(* CODESYS project MyRPIEtherCAT_2ESC.project

Project tree, tasks and I/O mapping:
  Device : CODESYS Control for Raspberry Pi SL, 3S - Smart Software Solutions GmbH, version 3.5.10.20
    application TestBlink
      libraries: Standard, * (System); Util, * (System)
      task MainTask (cyclic, interval 4000 µs, priority 0) calls EtherCAT_Master.EtherCAT_Task [EtherCAT_Master.EtherCAT_Task], PLC_PRG
      program PLC_PRG [LD]
      global variables GVL
    SoftMotion General Axis Pool
    I²C
    SPI
    GPIOs_A_B : GPIOs A/B, 3S - Smart Software Solutions GmbH, version 1.1.1.10
        output TestBlink.GVL.MASTER_LED1 : BOOL  // digital outputs (GPIO0..GPIO31).Bit17
        output TestBlink.GVL.MASTER_LED2 : BOOL  // digital outputs (GPIO0..GPIO31).Bit27
        unmapped channels: digital inputs (GPIO0..GPIO31), digital outputs (GPIO0..GPIO31)
    Onewire
    Camera device
      <Empty>
    EtherCAT_Master : EtherCAT Master, 3S - Smart Software Solutions GmbH, version 3.5.10.0
        settings: SrcAddress1 = 47143; SrcAddress2 = 3943328884
      XMC_ESC : XMC_ESC, Bahoza, order no. XMC_ESC, version Revision=16#00000000
          settings: StationAlias = 1001; Optional = False; DC sync0 cycletime = 4000; DC sync1 cycletime = 4000; RxTxPdo.NumberofExcludes = 0; RxTxPdo.NumberofEntries = 12; RxTxPdo.Index = 16#1600; RxTxPdo.Fixed = True; RxTxPdo.Mandatory = True; RxTxPdo.Virtual = False; RxTxPdo.Sm = 2; RxTxPdo.Su = 2; RxTxPdo.Name = 'OUT_GENERIC process data mapping'; RxTxPdo.DependOnSlot = False; RxTxPdo.DependOnSlotGroup = False; RxTxPdo.OverwrittenByModule = False; OUT_GEN_INT1.Index = 16#7000; OUT_GEN_INT1.SubIndex = 1; OUT_GEN_INT1.Size = 16; OUT_GEN_INT1.Offset = 0; OUT_GEN_INT1.DependOnSlot = False; OUT_GEN_INT1.DependOnSlotGroup = False; OUT_GEN_INT2.Index = 16#7000; OUT_GEN_INT2.SubIndex = 2; OUT_GEN_INT2.Size = 16; OUT_GEN_INT2.Offset = 0; OUT_GEN_INT2.DependOnSlot = False; OUT_GEN_INT2.DependOnSlotGroup = False; OUT_GEN_INT3.Index = 16#7000; OUT_GEN_INT3.SubIndex = 3; OUT_GEN_INT3.Size = 16; OUT_GEN_INT3.Offset = 0; OUT_GEN_INT3.DependOnSlot = False; OUT_GEN_INT3.DependOnSlotGroup = False; OUT_GEN_INT4.Index = 16#7000; OUT_GEN_INT4.SubIndex = 4; OUT_GEN_INT4.Size = 16; OUT_GEN_INT4.Offset = 0; OUT_GEN_INT4.DependOnSlot = False; OUT_GEN_INT4.DependOnSlotGroup = False;
            OUT_GEN_Bit1.Index = 16#7000; OUT_GEN_Bit1.SubIndex = 5; OUT_GEN_Bit1.Size = 1; OUT_GEN_Bit1.Offset = 0; OUT_GEN_Bit1.DependOnSlot = False; OUT_GEN_Bit1.DependOnSlotGroup = False; OUT_GEN_Bit2.Index = 16#7000; OUT_GEN_Bit2.SubIndex = 6; OUT_GEN_Bit2.Size = 1; OUT_GEN_Bit2.Offset = 0; OUT_GEN_Bit2.DependOnSlot = False; OUT_GEN_Bit2.DependOnSlotGroup = False; OUT_GEN_Bit3.Index = 16#7000; OUT_GEN_Bit3.SubIndex = 7; OUT_GEN_Bit3.Size = 1; OUT_GEN_Bit3.Offset = 0; OUT_GEN_Bit3.DependOnSlot = False; OUT_GEN_Bit3.DependOnSlotGroup = False; OUT_GEN_Bit4.Index = 16#7000; OUT_GEN_Bit4.SubIndex = 8; OUT_GEN_Bit4.Size = 1; OUT_GEN_Bit4.Offset = 0; OUT_GEN_Bit4.DependOnSlot = False; OUT_GEN_Bit4.DependOnSlotGroup = False; OUT_GEN_Bit5.Index = 16#7000; OUT_GEN_Bit5.SubIndex = 9; OUT_GEN_Bit5.Size = 1; OUT_GEN_Bit5.Offset = 0; OUT_GEN_Bit5.DependOnSlot = False; OUT_GEN_Bit5.DependOnSlotGroup = False; OUT_GEN_Bit6.Index = 16#7000; OUT_GEN_Bit6.SubIndex = 10; OUT_GEN_Bit6.Size = 1; OUT_GEN_Bit6.Offset = 0; OUT_GEN_Bit6.DependOnSlot = False; OUT_GEN_Bit6.DependOnSlotGroup = False; OUT_GEN_Bit7.Index = 16#7000; OUT_GEN_Bit7.SubIndex = 11; OUT_GEN_Bit7.Size = 1; OUT_GEN_Bit7.Offset = 0;
            OUT_GEN_Bit7.DependOnSlot = False; OUT_GEN_Bit7.DependOnSlotGroup = False; OUT_GEN_Bit8.Index = 16#7000; OUT_GEN_Bit8.SubIndex = 12; OUT_GEN_Bit8.Size = 1; OUT_GEN_Bit8.Offset = 0; OUT_GEN_Bit8.DependOnSlot = False; OUT_GEN_Bit8.DependOnSlotGroup = False; RxTxPdo.NumberofExcludes = 0; RxTxPdo.NumberofEntries = 12; RxTxPdo.Index = 16#1A00; RxTxPdo.Fixed = True; RxTxPdo.Mandatory = True; RxTxPdo.Virtual = False; RxTxPdo.Sm = 3; RxTxPdo.Su = 3; RxTxPdo.Name = 'IN_GENERIC process data mapping'; RxTxPdo.DependOnSlot = False; RxTxPdo.DependOnSlotGroup = False; RxTxPdo.OverwrittenByModule = False; IN_GEN_INT1.Index = 16#6000; IN_GEN_INT1.SubIndex = 1; IN_GEN_INT1.Size = 16; IN_GEN_INT1.Offset = 0; IN_GEN_INT1.DependOnSlot = False; IN_GEN_INT1.DependOnSlotGroup = False; IN_GEN_INT2.Index = 16#6000; IN_GEN_INT2.SubIndex = 2; IN_GEN_INT2.Size = 16; IN_GEN_INT2.Offset = 0; IN_GEN_INT2.DependOnSlot = False; IN_GEN_INT2.DependOnSlotGroup = False; IN_GEN_INT3.Index = 16#6000; IN_GEN_INT3.SubIndex = 3; IN_GEN_INT3.Size = 16; IN_GEN_INT3.Offset = 0; IN_GEN_INT3.DependOnSlot = False; IN_GEN_INT3.DependOnSlotGroup = False; IN_GEN_INT4.Index = 16#6000; IN_GEN_INT4.SubIndex = 4;
            IN_GEN_INT4.Size = 16; IN_GEN_INT4.Offset = 0; IN_GEN_INT4.DependOnSlot = False; IN_GEN_INT4.DependOnSlotGroup = False; IN_GEN_Bit1.Index = 16#6000; IN_GEN_Bit1.SubIndex = 5; IN_GEN_Bit1.Size = 1; IN_GEN_Bit1.Offset = 0; IN_GEN_Bit1.DependOnSlot = False; IN_GEN_Bit1.DependOnSlotGroup = False; IN_GEN_Bit2.Index = 16#6000; IN_GEN_Bit2.SubIndex = 6; IN_GEN_Bit2.Size = 1; IN_GEN_Bit2.Offset = 0; IN_GEN_Bit2.DependOnSlot = False; IN_GEN_Bit2.DependOnSlotGroup = False; IN_GEN_Bit3.Index = 16#6000; IN_GEN_Bit3.SubIndex = 7; IN_GEN_Bit3.Size = 1; IN_GEN_Bit3.Offset = 0; IN_GEN_Bit3.DependOnSlot = False; IN_GEN_Bit3.DependOnSlotGroup = False; IN_GEN_Bit4.Index = 16#6000; IN_GEN_Bit4.SubIndex = 8; IN_GEN_Bit4.Size = 1; IN_GEN_Bit4.Offset = 0; IN_GEN_Bit4.DependOnSlot = False; IN_GEN_Bit4.DependOnSlotGroup = False; IN_GEN_Bit5.Index = 16#6000; IN_GEN_Bit5.SubIndex = 9; IN_GEN_Bit5.Size = 1; IN_GEN_Bit5.Offset = 0; IN_GEN_Bit5.DependOnSlot = False; IN_GEN_Bit5.DependOnSlotGroup = False; IN_GEN_Bit6.Index = 16#6000; IN_GEN_Bit6.SubIndex = 10; IN_GEN_Bit6.Size = 1; IN_GEN_Bit6.Offset = 0; IN_GEN_Bit6.DependOnSlot = False; IN_GEN_Bit6.DependOnSlotGroup = False;
            IN_GEN_Bit7.Index = 16#6000; IN_GEN_Bit7.SubIndex = 11; IN_GEN_Bit7.Size = 1; IN_GEN_Bit7.Offset = 0; IN_GEN_Bit7.DependOnSlot = False; IN_GEN_Bit7.DependOnSlotGroup = False; IN_GEN_Bit8.Index = 16#6000; IN_GEN_Bit8.SubIndex = 12; IN_GEN_Bit8.Size = 1; IN_GEN_Bit8.Offset = 0; IN_GEN_Bit8.DependOnSlot = False; IN_GEN_Bit8.DependOnSlotGroup = False; OUT_GEN_INT1.Name = 'OUT_GEN_INT1'; OUT_GEN_INT1.DataType = 'UINT'; OUT_GEN_INT1.Default = ''; OUT_GEN_INT1.Comment = ''; OUT_GEN_INT2.Name = 'OUT_GEN_INT2'; OUT_GEN_INT2.DataType = 'UINT'; OUT_GEN_INT2.Default = ''; OUT_GEN_INT2.Comment = ''; OUT_GEN_INT3.Name = 'OUT_GEN_INT3'; OUT_GEN_INT3.DataType = 'UINT'; OUT_GEN_INT3.Default = ''; OUT_GEN_INT3.Comment = ''; OUT_GEN_INT4.Name = 'OUT_GEN_INT4'; OUT_GEN_INT4.DataType = 'UINT'; OUT_GEN_INT4.Default = ''; OUT_GEN_INT4.Comment = ''; OUT_GEN_Bit1.Name = 'OUT_GEN_Bit1'; OUT_GEN_Bit1.DataType = 'BIT'; OUT_GEN_Bit1.Default = ''; OUT_GEN_Bit1.Comment = ''; OUT_GEN_Bit2.Name = 'OUT_GEN_Bit2'; OUT_GEN_Bit2.DataType = 'BIT'; OUT_GEN_Bit2.Default = ''; OUT_GEN_Bit2.Comment = ''; OUT_GEN_Bit3.Name = 'OUT_GEN_Bit3'; OUT_GEN_Bit3.DataType = 'BIT'; OUT_GEN_Bit3.Default = ''; OUT_GEN_Bit3.Comment = '';
            OUT_GEN_Bit4.Name = 'OUT_GEN_Bit4'; OUT_GEN_Bit4.DataType = 'BIT'; OUT_GEN_Bit4.Default = ''; OUT_GEN_Bit4.Comment = ''; OUT_GEN_Bit5.Name = 'OUT_GEN_Bit5'; OUT_GEN_Bit5.DataType = 'BIT'; OUT_GEN_Bit5.Default = ''; OUT_GEN_Bit5.Comment = ''; OUT_GEN_Bit6.Name = 'OUT_GEN_Bit6'; OUT_GEN_Bit6.DataType = 'BIT'; OUT_GEN_Bit6.Default = ''; OUT_GEN_Bit6.Comment = ''; OUT_GEN_Bit7.Name = 'OUT_GEN_Bit7'; OUT_GEN_Bit7.DataType = 'BIT'; OUT_GEN_Bit7.Default = ''; OUT_GEN_Bit7.Comment = ''; OUT_GEN_Bit8.Name = 'OUT_GEN_Bit8'; OUT_GEN_Bit8.DataType = 'BIT'; OUT_GEN_Bit8.Default = ''; OUT_GEN_Bit8.Comment = ''; IN_GEN_INT1.Name = 'IN_GEN_INT1'; IN_GEN_INT1.DataType = 'UINT'; IN_GEN_INT1.Default = ''; IN_GEN_INT1.Comment = ''; IN_GEN_INT2.Name = 'IN_GEN_INT2'; IN_GEN_INT2.DataType = 'UINT'; IN_GEN_INT2.Default = ''; IN_GEN_INT2.Comment = ''; IN_GEN_INT3.Name = 'IN_GEN_INT3'; IN_GEN_INT3.DataType = 'UINT'; IN_GEN_INT3.Default = ''; IN_GEN_INT3.Comment = ''; IN_GEN_INT4.Name = 'IN_GEN_INT4'; IN_GEN_INT4.DataType = 'UINT'; IN_GEN_INT4.Default = ''; IN_GEN_INT4.Comment = ''; IN_GEN_Bit1.Name = 'IN_GEN_Bit1'; IN_GEN_Bit1.DataType = 'BIT'; IN_GEN_Bit1.Default = ''; IN_GEN_Bit1.Comment = '';
            IN_GEN_Bit2.Name = 'IN_GEN_Bit2'; IN_GEN_Bit2.DataType = 'BIT'; IN_GEN_Bit2.Default = ''; IN_GEN_Bit2.Comment = ''; IN_GEN_Bit3.Name = 'IN_GEN_Bit3'; IN_GEN_Bit3.DataType = 'BIT'; IN_GEN_Bit3.Default = ''; IN_GEN_Bit3.Comment = ''; IN_GEN_Bit4.Name = 'IN_GEN_Bit4'; IN_GEN_Bit4.DataType = 'BIT'; IN_GEN_Bit4.Default = ''; IN_GEN_Bit4.Comment = ''; IN_GEN_Bit5.Name = 'IN_GEN_Bit5'; IN_GEN_Bit5.DataType = 'BIT'; IN_GEN_Bit5.Default = ''; IN_GEN_Bit5.Comment = ''; IN_GEN_Bit6.Name = 'IN_GEN_Bit6'; IN_GEN_Bit6.DataType = 'BIT'; IN_GEN_Bit6.Default = ''; IN_GEN_Bit6.Comment = ''; IN_GEN_Bit7.Name = 'IN_GEN_Bit7'; IN_GEN_Bit7.DataType = 'BIT'; IN_GEN_Bit7.Default = ''; IN_GEN_Bit7.Comment = ''; IN_GEN_Bit8.Name = 'IN_GEN_Bit8'; IN_GEN_Bit8.DataType = 'BIT'; IN_GEN_Bit8.Default = ''; IN_GEN_Bit8.Comment = ''
          output TestBlink.GVL.SLAVE1_LED1 : BIT  // OUT_GEN_Bit1
          input  TestBlink.GVL.SLAVE1_BTN1 : BIT  // IN_GEN_Bit1
          unmapped channels: OUT_GEN_INT1, OUT_GEN_INT2, OUT_GEN_INT3, OUT_GEN_INT4, OUT_GEN_Bit2, OUT_GEN_Bit3, OUT_GEN_Bit4, OUT_GEN_Bit5, OUT_GEN_Bit6, OUT_GEN_Bit7, OUT_GEN_Bit8, IN_GEN_INT1, IN_GEN_INT2, IN_GEN_INT3, IN_GEN_INT4, IN_GEN_Bit2, IN_GEN_Bit3, IN_GEN_Bit4, IN_GEN_Bit5, IN_GEN_Bit6, IN_GEN_Bit7, IN_GEN_Bit8
      XMC_ESC_2 : XMC_ESC, Bahoza, order no. XMC_ESC, version Revision=16#00000000
          settings: DC sync0 cycletime = 4000; DC sync1 cycletime = 4000; RxTxPdo.NumberofExcludes = 0; RxTxPdo.NumberofEntries = 12; RxTxPdo.Index = 16#1600; RxTxPdo.Fixed = True; RxTxPdo.Mandatory = True; RxTxPdo.Virtual = False; RxTxPdo.Sm = 2; RxTxPdo.Su = 2; RxTxPdo.Name = 'OUT_GENERIC process data mapping'; RxTxPdo.DependOnSlot = False; RxTxPdo.DependOnSlotGroup = False; RxTxPdo.OverwrittenByModule = False; OUT_GEN_INT1.Index = 16#7000; OUT_GEN_INT1.SubIndex = 1; OUT_GEN_INT1.Size = 16; OUT_GEN_INT1.Offset = 0; OUT_GEN_INT1.DependOnSlot = False; OUT_GEN_INT1.DependOnSlotGroup = False; OUT_GEN_INT2.Index = 16#7000; OUT_GEN_INT2.SubIndex = 2; OUT_GEN_INT2.Size = 16; OUT_GEN_INT2.Offset = 0; OUT_GEN_INT2.DependOnSlot = False; OUT_GEN_INT2.DependOnSlotGroup = False; OUT_GEN_INT3.Index = 16#7000; OUT_GEN_INT3.SubIndex = 3; OUT_GEN_INT3.Size = 16; OUT_GEN_INT3.Offset = 0; OUT_GEN_INT3.DependOnSlot = False; OUT_GEN_INT3.DependOnSlotGroup = False; OUT_GEN_INT4.Index = 16#7000; OUT_GEN_INT4.SubIndex = 4; OUT_GEN_INT4.Size = 16; OUT_GEN_INT4.Offset = 0; OUT_GEN_INT4.DependOnSlot = False; OUT_GEN_INT4.DependOnSlotGroup = False; OUT_GEN_Bit1.Index = 16#7000; OUT_GEN_Bit1.SubIndex = 5;
            OUT_GEN_Bit1.Size = 1; OUT_GEN_Bit1.Offset = 0; OUT_GEN_Bit1.DependOnSlot = False; OUT_GEN_Bit1.DependOnSlotGroup = False; OUT_GEN_Bit2.Index = 16#7000; OUT_GEN_Bit2.SubIndex = 6; OUT_GEN_Bit2.Size = 1; OUT_GEN_Bit2.Offset = 0; OUT_GEN_Bit2.DependOnSlot = False; OUT_GEN_Bit2.DependOnSlotGroup = False; OUT_GEN_Bit3.Index = 16#7000; OUT_GEN_Bit3.SubIndex = 7; OUT_GEN_Bit3.Size = 1; OUT_GEN_Bit3.Offset = 0; OUT_GEN_Bit3.DependOnSlot = False; OUT_GEN_Bit3.DependOnSlotGroup = False; OUT_GEN_Bit4.Index = 16#7000; OUT_GEN_Bit4.SubIndex = 8; OUT_GEN_Bit4.Size = 1; OUT_GEN_Bit4.Offset = 0; OUT_GEN_Bit4.DependOnSlot = False; OUT_GEN_Bit4.DependOnSlotGroup = False; OUT_GEN_Bit5.Index = 16#7000; OUT_GEN_Bit5.SubIndex = 9; OUT_GEN_Bit5.Size = 1; OUT_GEN_Bit5.Offset = 0; OUT_GEN_Bit5.DependOnSlot = False; OUT_GEN_Bit5.DependOnSlotGroup = False; OUT_GEN_Bit6.Index = 16#7000; OUT_GEN_Bit6.SubIndex = 10; OUT_GEN_Bit6.Size = 1; OUT_GEN_Bit6.Offset = 0; OUT_GEN_Bit6.DependOnSlot = False; OUT_GEN_Bit6.DependOnSlotGroup = False; OUT_GEN_Bit7.Index = 16#7000; OUT_GEN_Bit7.SubIndex = 11; OUT_GEN_Bit7.Size = 1; OUT_GEN_Bit7.Offset = 0; OUT_GEN_Bit7.DependOnSlot = False; OUT_GEN_Bit7.DependOnSlotGroup = False;
            OUT_GEN_Bit8.Index = 16#7000; OUT_GEN_Bit8.SubIndex = 12; OUT_GEN_Bit8.Size = 1; OUT_GEN_Bit8.Offset = 0; OUT_GEN_Bit8.DependOnSlot = False; OUT_GEN_Bit8.DependOnSlotGroup = False; RxTxPdo.NumberofExcludes = 0; RxTxPdo.NumberofEntries = 12; RxTxPdo.Index = 16#1A00; RxTxPdo.Fixed = True; RxTxPdo.Mandatory = True; RxTxPdo.Virtual = False; RxTxPdo.Sm = 3; RxTxPdo.Su = 3; RxTxPdo.Name = 'IN_GENERIC process data mapping'; RxTxPdo.DependOnSlot = False; RxTxPdo.DependOnSlotGroup = False; RxTxPdo.OverwrittenByModule = False; IN_GEN_INT1.Index = 16#6000; IN_GEN_INT1.SubIndex = 1; IN_GEN_INT1.Size = 16; IN_GEN_INT1.Offset = 0; IN_GEN_INT1.DependOnSlot = False; IN_GEN_INT1.DependOnSlotGroup = False; IN_GEN_INT2.Index = 16#6000; IN_GEN_INT2.SubIndex = 2; IN_GEN_INT2.Size = 16; IN_GEN_INT2.Offset = 0; IN_GEN_INT2.DependOnSlot = False; IN_GEN_INT2.DependOnSlotGroup = False; IN_GEN_INT3.Index = 16#6000; IN_GEN_INT3.SubIndex = 3; IN_GEN_INT3.Size = 16; IN_GEN_INT3.Offset = 0; IN_GEN_INT3.DependOnSlot = False; IN_GEN_INT3.DependOnSlotGroup = False; IN_GEN_INT4.Index = 16#6000; IN_GEN_INT4.SubIndex = 4; IN_GEN_INT4.Size = 16; IN_GEN_INT4.Offset = 0;
            IN_GEN_INT4.DependOnSlot = False; IN_GEN_INT4.DependOnSlotGroup = False; IN_GEN_Bit1.Index = 16#6000; IN_GEN_Bit1.SubIndex = 5; IN_GEN_Bit1.Size = 1; IN_GEN_Bit1.Offset = 0; IN_GEN_Bit1.DependOnSlot = False; IN_GEN_Bit1.DependOnSlotGroup = False; IN_GEN_Bit2.Index = 16#6000; IN_GEN_Bit2.SubIndex = 6; IN_GEN_Bit2.Size = 1; IN_GEN_Bit2.Offset = 0; IN_GEN_Bit2.DependOnSlot = False; IN_GEN_Bit2.DependOnSlotGroup = False; IN_GEN_Bit3.Index = 16#6000; IN_GEN_Bit3.SubIndex = 7; IN_GEN_Bit3.Size = 1; IN_GEN_Bit3.Offset = 0; IN_GEN_Bit3.DependOnSlot = False; IN_GEN_Bit3.DependOnSlotGroup = False; IN_GEN_Bit4.Index = 16#6000; IN_GEN_Bit4.SubIndex = 8; IN_GEN_Bit4.Size = 1; IN_GEN_Bit4.Offset = 0; IN_GEN_Bit4.DependOnSlot = False; IN_GEN_Bit4.DependOnSlotGroup = False; IN_GEN_Bit5.Index = 16#6000; IN_GEN_Bit5.SubIndex = 9; IN_GEN_Bit5.Size = 1; IN_GEN_Bit5.Offset = 0; IN_GEN_Bit5.DependOnSlot = False; IN_GEN_Bit5.DependOnSlotGroup = False; IN_GEN_Bit6.Index = 16#6000; IN_GEN_Bit6.SubIndex = 10; IN_GEN_Bit6.Size = 1; IN_GEN_Bit6.Offset = 0; IN_GEN_Bit6.DependOnSlot = False; IN_GEN_Bit6.DependOnSlotGroup = False; IN_GEN_Bit7.Index = 16#6000; IN_GEN_Bit7.SubIndex = 11;
            IN_GEN_Bit7.Size = 1; IN_GEN_Bit7.Offset = 0; IN_GEN_Bit7.DependOnSlot = False; IN_GEN_Bit7.DependOnSlotGroup = False; IN_GEN_Bit8.Index = 16#6000; IN_GEN_Bit8.SubIndex = 12; IN_GEN_Bit8.Size = 1; IN_GEN_Bit8.Offset = 0; IN_GEN_Bit8.DependOnSlot = False; IN_GEN_Bit8.DependOnSlotGroup = False; OUT_GEN_INT1.Name = 'OUT_GEN_INT1'; OUT_GEN_INT1.DataType = 'UINT'; OUT_GEN_INT1.Default = ''; OUT_GEN_INT1.Comment = ''; OUT_GEN_INT2.Name = 'OUT_GEN_INT2'; OUT_GEN_INT2.DataType = 'UINT'; OUT_GEN_INT2.Default = ''; OUT_GEN_INT2.Comment = ''; OUT_GEN_INT3.Name = 'OUT_GEN_INT3'; OUT_GEN_INT3.DataType = 'UINT'; OUT_GEN_INT3.Default = ''; OUT_GEN_INT3.Comment = ''; OUT_GEN_INT4.Name = 'OUT_GEN_INT4'; OUT_GEN_INT4.DataType = 'UINT'; OUT_GEN_INT4.Default = ''; OUT_GEN_INT4.Comment = ''; OUT_GEN_Bit1.Name = 'OUT_GEN_Bit1'; OUT_GEN_Bit1.DataType = 'BIT'; OUT_GEN_Bit1.Default = ''; OUT_GEN_Bit1.Comment = ''; OUT_GEN_Bit2.Name = 'OUT_GEN_Bit2'; OUT_GEN_Bit2.DataType = 'BIT'; OUT_GEN_Bit2.Default = ''; OUT_GEN_Bit2.Comment = ''; OUT_GEN_Bit3.Name = 'OUT_GEN_Bit3'; OUT_GEN_Bit3.DataType = 'BIT'; OUT_GEN_Bit3.Default = ''; OUT_GEN_Bit3.Comment = ''; OUT_GEN_Bit4.Name = 'OUT_GEN_Bit4'; OUT_GEN_Bit4.DataType = 'BIT';
            OUT_GEN_Bit4.Default = ''; OUT_GEN_Bit4.Comment = ''; OUT_GEN_Bit5.Name = 'OUT_GEN_Bit5'; OUT_GEN_Bit5.DataType = 'BIT'; OUT_GEN_Bit5.Default = ''; OUT_GEN_Bit5.Comment = ''; OUT_GEN_Bit6.Name = 'OUT_GEN_Bit6'; OUT_GEN_Bit6.DataType = 'BIT'; OUT_GEN_Bit6.Default = ''; OUT_GEN_Bit6.Comment = ''; OUT_GEN_Bit7.Name = 'OUT_GEN_Bit7'; OUT_GEN_Bit7.DataType = 'BIT'; OUT_GEN_Bit7.Default = ''; OUT_GEN_Bit7.Comment = ''; OUT_GEN_Bit8.Name = 'OUT_GEN_Bit8'; OUT_GEN_Bit8.DataType = 'BIT'; OUT_GEN_Bit8.Default = ''; OUT_GEN_Bit8.Comment = ''; IN_GEN_INT1.Name = 'IN_GEN_INT1'; IN_GEN_INT1.DataType = 'UINT'; IN_GEN_INT1.Default = ''; IN_GEN_INT1.Comment = ''; IN_GEN_INT2.Name = 'IN_GEN_INT2'; IN_GEN_INT2.DataType = 'UINT'; IN_GEN_INT2.Default = ''; IN_GEN_INT2.Comment = ''; IN_GEN_INT3.Name = 'IN_GEN_INT3'; IN_GEN_INT3.DataType = 'UINT'; IN_GEN_INT3.Default = ''; IN_GEN_INT3.Comment = ''; IN_GEN_INT4.Name = 'IN_GEN_INT4'; IN_GEN_INT4.DataType = 'UINT'; IN_GEN_INT4.Default = ''; IN_GEN_INT4.Comment = ''; IN_GEN_Bit1.Name = 'IN_GEN_Bit1'; IN_GEN_Bit1.DataType = 'BIT'; IN_GEN_Bit1.Default = ''; IN_GEN_Bit1.Comment = ''; IN_GEN_Bit2.Name = 'IN_GEN_Bit2'; IN_GEN_Bit2.DataType = 'BIT';
            IN_GEN_Bit2.Default = ''; IN_GEN_Bit2.Comment = ''; IN_GEN_Bit3.Name = 'IN_GEN_Bit3'; IN_GEN_Bit3.DataType = 'BIT'; IN_GEN_Bit3.Default = ''; IN_GEN_Bit3.Comment = ''; IN_GEN_Bit4.Name = 'IN_GEN_Bit4'; IN_GEN_Bit4.DataType = 'BIT'; IN_GEN_Bit4.Default = ''; IN_GEN_Bit4.Comment = ''; IN_GEN_Bit5.Name = 'IN_GEN_Bit5'; IN_GEN_Bit5.DataType = 'BIT'; IN_GEN_Bit5.Default = ''; IN_GEN_Bit5.Comment = ''; IN_GEN_Bit6.Name = 'IN_GEN_Bit6'; IN_GEN_Bit6.DataType = 'BIT'; IN_GEN_Bit6.Default = ''; IN_GEN_Bit6.Comment = ''; IN_GEN_Bit7.Name = 'IN_GEN_Bit7'; IN_GEN_Bit7.DataType = 'BIT'; IN_GEN_Bit7.Default = ''; IN_GEN_Bit7.Comment = ''; IN_GEN_Bit8.Name = 'IN_GEN_Bit8'; IN_GEN_Bit8.DataType = 'BIT'; IN_GEN_Bit8.Default = ''; IN_GEN_Bit8.Comment = ''
          output TestBlink.GVL.SLAVE2_LED1 : BIT  // OUT_GEN_Bit1
          input  TestBlink.GVL.SLAVE2_BTN1 : BIT  // IN_GEN_Bit1
          unmapped channels: OUT_GEN_INT1, OUT_GEN_INT2, OUT_GEN_INT3, OUT_GEN_INT4, OUT_GEN_Bit2, OUT_GEN_Bit3, OUT_GEN_Bit4, OUT_GEN_Bit5, OUT_GEN_Bit6, OUT_GEN_Bit7, OUT_GEN_Bit8, IN_GEN_INT1, IN_GEN_INT2, IN_GEN_INT3, IN_GEN_INT4, IN_GEN_Bit2, IN_GEN_Bit3, IN_GEN_Bit4, IN_GEN_Bit5, IN_GEN_Bit6, IN_GEN_Bit7, IN_GEN_Bit8
*)

// Device/TestBlink/GVL
{attribute 'qualified_only'}
VAR_GLOBAL
	MASTER_LED1: BOOL;
	MASTER_LED2: BOOL;
	SLAVE1_LED1: BOOL;
	SLAVE1_BTN1: BOOL;
	SLAVE2_LED1: BOOL;
	SLAVE2_BTN1: BOOL;
END_VAR

// Device/TestBlink/PLC_PRG
PROGRAM PLC_PRG
VAR
	Test_ON: BOOL;
	Test_OUT: BOOL;
	EthBlink1: BLINK := (TIMELOW := TIME#500ms, TIMEHIGH := TIME#500ms);
	EthBlink2: BLINK := (TIMELOW := TIME#1s0ms, TIMEHIGH := TIME#1s0ms);
END_VAR

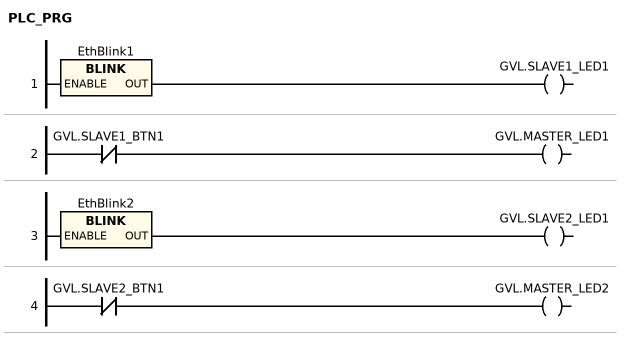
// NETWORK 1
EthBlink1(ENABLE := TRUE); // BLINK
GVL.SLAVE1_LED1 := EthBlink1.OUT;

// NETWORK 2
GVL.MASTER_LED1 := NOT GVL.SLAVE1_BTN1;

// NETWORK 3
EthBlink2(ENABLE := TRUE); // BLINK
GVL.SLAVE2_LED1 := EthBlink2.OUT;

// NETWORK 4
GVL.MASTER_LED2 := NOT GVL.SLAVE2_BTN1;

END_PROGRAM
